Yaskawa INFORM job: OK_R2_O34(P)(180,90)OKKR.JBI

/JOB
//NAME OK_R2_O34(P)(180,90)OKKR
///FOLDERNAME X4
//POS
///NPOS 169,169,169,10,0,0
///TOOL 0
///POSTYPE PULSE
///PULSE
C00000=-166198,-138144,-82480,-6370,52509,85895
C00001=-166198,-138144,-82480,-6370,52509,85895
C00002=-181117,-122681,-70821,-2391,52511,79976
C00003=-181117,-121299,-68978,-2404,52087,79986
C00004=-181117,-122681,-70821,-2391,52511,79976
C00005=-189750,-118853,-70881,1473,64532,76480
C00006=-190053,-120746,-70880,1514,63564,76360
C00007=-189750,-118853,-70881,1473,64532,76480
C00008=-189574,-119616,-72884,1448,65370,76553
C00009=-189152,-121343,-77794,1387,67496,76728
C00010=-185679,-117174,-91161,1016,77811,78037
C00011=-185951,-117066,-86971,1049,75292,77923
C00012=-186063,-116900,-85242,1063,74315,77875
C00013=-185963,-114657,-82563,1057,73818,77905
C00014=-186063,-116900,-85242,1063,74315,77875
C00015=-189745,-129542,-86508,1430,68655,76533
C00016=-190220,-131942,-86638,1484,67510,76354
C00017=-189745,-129542,-86508,1430,68655,76533
C00018=-189571,-130130,-88400,1406,69515,76605
C00019=-189152,-131370,-93030,1352,71719,76776
C00020=-186714,-125767,-101679,2828,70067,77519
C00021=-186815,-124081,-96932,2888,68019,77434
C00022=-186348,-121871,-95196,2777,68068,77605
C00023=-186348,-120596,-92866,2792,67290,77587
C00024=-186348,-121871,-95196,2777,68068,77605
C00025=-189400,-136727,-97452,3651,61954,76311
C00026=-189193,-138074,-96714,3640,60801,76351
C00027=-189400,-136727,-97452,3651,61954,76311
C00028=-188527,-137172,-98533,3430,62352,76650
C00029=-188394,-140146,-103663,3351,63973,76748
C00030=-205862,-111673,-97339,6868,75787,70984
C00031=-186550,-124540,-97192,2829,67933,77528
C00032=-186590,-123775,-95257,2853,67137,77494
C00033=-186478,-121948,-93528,2830,67009,77531
C00034=-186590,-123775,-95257,2853,67137,77494
C00035=-188399,-134884,-95960,3412,61939,76686
C00036=-188879,-137801,-96233,3570,60632,76465
C00037=-188399,-134884,-95960,3412,61939,76686
C00038=-188346,-136077,-98025,3379,62594,76725
C00039=-188215,-138975,-103137,3302,64243,76822
C00040=-204668,-125654,-103075,12731,76819,72583
C00041=-192085,-108894,-77492,34918,79459,78781
C00042=-188431,-109256,-74124,35205,76110,79208
C00043=-186907,-109255,-72716,35331,74778,79404
C00044=-186693,-106850,-70345,35364,74503,79405
C00045=-186907,-109255,-72716,35331,74778,79404
C00046=-188549,-120012,-73127,36179,71120,77489
C00047=-189163,-122031,-72881,36386,70400,76982
C00048=-188549,-120012,-73127,36179,71120,77489
C00049=-190319,-120259,-74660,35963,72503,77227
C00050=-194524,-120520,-78356,35450,75955,76649
C00051=-198919,-109995,-61190,42638,67655,70810
C00052=-190285,-110618,-59420,40336,62273,73169
C00053=-188753,-109213,-57500,40420,61811,73628
C00054=-188509,-106588,-54755,40535,61445,73582
C00055=-188753,-109213,-57500,40420,61811,73628
C00056=-188387,-108235,-55987,37151,67409,76240
C00057=-189079,-110340,-56039,37365,66843,75742
C00058=-188387,-108235,-55987,37151,67409,76240
C00059=-190169,-108675,-57643,36861,68766,75986
C00060=-194403,-109476,-61648,36169,72132,75416
C00061=-225594,-162129,-113087,31828,88019,68030
C00062=-139895,-75891,-115387,-4844,89852,-32669
C00063=-106959,-65294,-90716,-19296,63371,-70213
C00064=-120633,-142199,-78464,-12,37387,-81752
C00065=-120609,-138941,-73010,-25,35704,-81740
C00066=-120602,-137609,-70801,-31,35029,-81735
C00067=-120604,-135014,-68605,-30,35012,-81736
C00068=-120602,-137609,-70801,-31,35029,-81735
C00069=-120446,-129838,-71958,-24,53874,-81685
C00070=-120438,-131177,-71579,-25,52953,-81682
C00071=-120446,-129838,-71958,-24,53874,-81685
C00072=-131738,-132228,-73452,8067,51560,-87163
C00073=-139177,-145158,-85992,13671,51481,-90607
C00074=-120880,-115298,-90682,38,78334,-81839
C00075=-120874,-115322,-86545,38,75775,-81838
C00076=-120876,-117328,-85486,38,74093,-81838
C00077=-120874,-115144,-83188,38,73801,-81838
C00078=-120876,-117328,-85486,38,74093,-81838
C00079=-120239,-131127,-87989,-18,68542,-81617
C00080=-120200,-135397,-88149,-23,66446,-81603
C00081=-120239,-131127,-87989,-18,68542,-81617
C00082=-120250,-131705,-89876,-17,69407,-81621
C00083=-120275,-132914,-94493,-15,71627,-81630
C00084=-120870,-123802,-101141,29,70454,-81834
C00085=-120864,-122259,-96439,28,68353,-81832
C00086=-120864,-123447,-95607,27,67230,-81833
C00087=-120862,-121131,-93340,27,67025,-81832
C00088=-120864,-123447,-95607,27,67230,-81833
C00089=-122761,-109093,-90522,1639,82538,-82345
C00090=-122816,-111754,-90455,1648,81130,-82381
C00091=-122761,-109093,-90522,1639,82538,-82345
C00092=-120406,-97391,-87876,-7,91529,-81675
C00093=-120406,-100930,-93432,-13,91808,-81675
C00094=-120586,-133914,-102382,9547,85095,-1839
C00095=-120585,-130719,-97494,9563,83747,-1942
C00096=-121451,-155216,-100429,10564,64059,-3872
C00097=-120574,-132034,-95782,9591,82039,-2069
C00098=-120583,-131496,-97319,9570,83246,-1979
C00099=-101302,-152747,-99963,8345,62763,3312
C00100=-120585,-128649,-94311,19028,83925,-4078
C00101=-120586,-131726,-99006,19000,85165,-3884
C00102=-120584,-126515,-91053,9592,81967,-2078
C00103=-120583,-123236,-86048,9622,80591,-2184
C00104=-121323,-131959,-83025,11198,58345,-4395
C00105=-120572,-124091,-84174,9663,79018,-2303
C00106=-120581,-123849,-85824,9632,80143,-2218
C00107=-103313,-130201,-82619,7208,57008,2414
C00108=-104272,-134854,-85867,7955,57176,1910
C00109=-120583,-124266,-87596,19086,82143,-4357
C00110=-121487,-140866,-77356,12448,52400,-5292
C00111=-120447,-141800,-70609,13740,42943,-6005
C00112=-120557,-138216,-68435,13384,45148,-5776
C00113=-120569,-112606,-67195,9826,74534,-2658
C00114=-120578,-112690,-68999,9781,75586,-2576
C00115=-93586,-136115,-68174,5406,43260,5492
C00116=-92921,-144795,-73490,5308,42038,5703
C00117=-124561,-133641,-73213,24753,58902,-8707
C00118=-106959,-65294,-90716,-19296,63371,-70213
C00119=-139895,-75891,-115387,-4844,89852,-32669
C00120=-225594,-162129,-113087,31828,88019,68030
C00121=-179306,-113082,-59158,46822,53733,18344
C00122=-185426,-123846,-62062,47213,53042,4581
C00123=-178966,-109306,-51351,46489,50599,6676
C00124=-174320,-104192,-54351,40123,55740,30099
C00125=-174328,-104480,-56277,39686,56549,30457
C00126=-160513,-108482,-51153,43765,42263,12341
C00127=-163416,-122959,-61489,45174,42800,10900
C00128=-171485,-113063,-58167,48901,53583,17150
C00129=-174246,-118964,-79181,37262,61787,32648
C00130=-175314,-125675,-85082,29507,69100,6827
C00131=-172538,-123885,-72027,36900,51897,2976
C00132=-174245,-116047,-71991,38244,59447,31724
C00133=-174254,-116050,-73753,37868,60313,32068
C00134=-155711,-121999,-71583,32332,45981,9052
C00135=-157559,-134878,-79454,33856,45162,7759
C00136=-184822,-140786,-87725,38201,57754,-504
C00137=-174185,-126575,-90838,36294,64403,33652
C00138=-184546,-129565,-98731,33104,80671,8257
C00139=-172470,-130384,-85545,34125,57897,8623
C00140=-174183,-124125,-83946,37166,61986,32753
C00141=-174193,-123890,-85598,36821,62909,33098
C00142=-156624,-128212,-85008,30161,52691,14183
C00143=-158543,-145659,-95435,31710,51171,12758
C00144=-172584,-141042,-104059,24276,66357,13202
C00145=-174271,-134419,-102558,-9435,85095,2061
C00146=-174282,-131199,-97661,-9450,83752,2158
C00147=-164002,-160404,-98949,-17577,58586,9036
C00148=-174285,-131975,-97483,-9458,83250,2195
C00149=-174277,-132508,-95944,-9478,82045,2290
C00150=-187249,-159818,-98857,-14082,54575,657
C00151=-174172,-139478,-100543,-16924,80978,4815
C00152=-174270,-132235,-99253,-18877,85281,4097
C00153=-174331,-126988,-91193,-9482,81954,2278
C00154=-155939,-119712,-87863,-13482,83832,9313
C00155=-158672,-128715,-82609,-15704,65966,9091
C00156=-174346,-124299,-85953,-9522,80133,2412
C00157=-174339,-124536,-84301,-9552,79010,2501
C00158=-176166,-130256,-82976,-13742,62349,3087
C00159=-165849,-135350,-93004,-16350,73762,7142
C00160=-174331,-124753,-87812,-18965,82235,4549
C00161=-174405,-116101,-74598,-9605,77388,2605
C00162=-166751,-128810,-77158,-12073,63289,6016
C00163=-170397,-124501,-65427,-14011,49451,5614
C00164=-174420,-113094,-69082,-9672,75561,2744
C00165=-174415,-113004,-67275,-9716,74511,2829
C00166=-190761,-123182,-65160,-8225,47369,-2619
C00167=-190350,-134813,-72783,-8527,46136,-2334
C00168=-168158,-141495,-72172,-29255,50267,11505
BC00000=196804,892977,1075175
BC00001=196804,892977,1075175
BC00002=196804,892977,1075175
BC00003=196804,892977,1075175
BC00004=196804,892977,1075175
BC00005=196804,892977,1075175
BC00006=196804,892977,1075175
BC00007=196804,892977,1075175
BC00008=196804,892977,1075175
BC00009=196804,892977,1075175
BC00010=223883,863738,1075175
BC00011=223883,863738,1075175
BC00012=223883,863738,1075175
BC00013=223883,863738,1075175
BC00014=223883,863738,1075175
BC00015=223883,863738,1075175
BC00016=223883,863738,1075175
BC00017=223883,863738,1075175
BC00018=223883,863738,1075175
BC00019=223883,863738,1075175
BC00020=258179,822666,1075175
BC00021=258179,822666,1075175
BC00022=258179,822666,1075175
BC00023=258179,822666,1075175
BC00024=258179,822666,1075175
BC00025=258179,822666,1075175
BC00026=258179,822666,1075175
BC00027=258179,822666,1075175
BC00028=258179,822666,1075175
BC00029=258179,822666,1075175
BC00030=349124,897467,1075175
BC00031=349124,897467,1075175
BC00032=349124,897467,1075175
BC00033=349124,897467,1075175
BC00034=349124,897467,1075175
BC00035=349124,897467,1075175
BC00036=349124,897467,1075175
BC00037=349124,897467,1075175
BC00038=349124,897467,1075175
BC00039=349124,897467,1075175
BC00040=330638,897048,1075175
BC00041=270427,895682,1075175
BC00042=270427,895682,1075175
BC00043=270427,895682,1075175
BC00044=270427,895682,1075175
BC00045=270427,895682,1075175
BC00046=270427,895682,1075175
BC00047=270427,895682,1075175
BC00048=270427,895682,1075175
BC00049=270427,895682,1075175
BC00050=270427,895682,1075175
BC00051=244019,926301,1075175
BC00052=244019,926301,1075175
BC00053=244019,926301,1075175
BC00054=244019,926301,1075175
BC00055=244019,926301,1075175
BC00056=244019,926301,1075175
BC00057=244019,926301,1075175
BC00058=244019,926301,1075175
BC00059=244019,926301,1075175
BC00060=244019,926301,1075175
BC00061=244019,926301,1075175
BC00062=284621,806624,1075175
BC00063=300201,760702,1075175
BC00064=369544,946445,1075175
BC00065=369544,946445,1075175
BC00066=369544,946445,1075175
BC00067=369544,946445,1075175
BC00068=369544,946445,1075175
BC00069=369544,946445,1075175
BC00070=369544,946445,1075175
BC00071=369544,946445,1075175
BC00072=369544,946445,1075175
BC00073=369544,946445,1075175
BC00074=370687,905748,1075175
BC00075=370687,905748,1075175
BC00076=370687,905748,1075175
BC00077=370687,905748,1075175
BC00078=370687,905748,1075175
BC00079=370687,905748,1075175
BC00080=370687,905748,1075175
BC00081=370687,905748,1075175
BC00082=370687,905748,1075175
BC00083=370687,905748,1075175
BC00084=370814,852872,1075175
BC00085=370814,852872,1075175
BC00086=370814,852872,1075175
BC00087=370814,852872,1075175
BC00088=370814,852872,1075175
BC00089=370814,852872,1075175
BC00090=370814,852872,1075175
BC00091=370814,852872,1075175
BC00092=370814,852872,1075175
BC00093=370814,852872,1075175
BC00094=333496,876256,1075175
BC00095=334875,878803,1075175
BC00096=335207,879415,1075175
BC00097=335427,879822,1075175
BC00098=335427,879822,1075175
BC00099=335207,879415,1075175
BC00100=332127,880440,1075175
BC00101=329407,878005,1075175
BC00102=333395,910749,1075175
BC00103=334774,913297,1075175
BC00104=335251,892678,1075175
BC00105=335326,914316,1075175
BC00106=335326,914316,1075175
BC00107=335251,892678,1075175
BC00108=335146,893402,1075175
BC00109=329306,912498,1075175
BC00110=333280,950895,1075175
BC00111=334659,953443,1075175
BC00112=334790,953685,1075175
BC00113=335211,954462,1075175
BC00114=335211,954462,1075175
BC00115=334790,953685,1075175
BC00116=334790,953685,1075175
BC00117=329191,952645,1075175
BC00118=300201,760702,1075175
BC00119=284621,806624,1075175
BC00120=244019,926301,1075175
BC00121=252810,904839,1075175
BC00122=251930,908762,1075175
BC00123=251930,908762,1075175
BC00124=251930,908762,1075175
BC00125=251930,908762,1075175
BC00126=251930,908762,1075175
BC00127=251930,908762,1075175
BC00128=250378,907547,1075175
BC00129=279615,874170,1075175
BC00130=278758,877989,1075175
BC00131=278758,877989,1075175
BC00132=278735,878093,1075175
BC00133=278735,878093,1075175
BC00134=278758,877989,1075175
BC00135=278758,877989,1075175
BC00136=278758,877989,1075175
BC00137=302654,847819,1075175
BC00138=301842,851437,1075175
BC00139=301842,851437,1075175
BC00140=301773,851742,1075175
BC00141=301773,851742,1075175
BC00142=301842,851437,1075175
BC00143=301842,851437,1075175
BC00144=301842,851437,1075175
BC00145=254856,848220,1075175
BC00146=252114,849302,1075175
BC00147=251037,849726,1075175
BC00148=251017,849734,1075175
BC00149=251017,849734,1075175
BC00150=251037,849726,1075175
BC00151=251037,849726,1075175
BC00152=256865,852098,1075175
BC00153=231817,874571,1075175
BC00154=231101,858363,1075175
BC00155=231101,858363,1075175
BC00156=227978,876085,1075175
BC00157=227978,876085,1075175
BC00158=231101,858363,1075175
BC00159=231101,858363,1075175
BC00160=233826,878449,1075175
BC00161=205012,905240,1075175
BC00162=209704,892317,1075175
BC00163=209704,892317,1075175
BC00164=201173,906754,1075175
BC00165=201173,906754,1075175
BC00166=209704,892317,1075175
BC00167=209704,892317,1075175
BC00168=207022,909118,1075175
EC00000=1596313,309153
EC00001=1596313,309153
EC00002=1596313,309153
EC00003=1596313,309153
EC00004=1596313,309153
EC00005=1596313,309153
EC00006=1596313,309153
EC00007=1596313,309153
EC00008=1596313,309153
EC00009=1596313,309153
EC00010=1596313,309153
EC00011=1596313,309153
EC00012=1596313,309153
EC00013=1596313,309153
EC00014=1596313,309153
EC00015=1596313,309153
EC00016=1596313,309153
EC00017=1596313,309153
EC00018=1596313,309153
EC00019=1596313,309153
EC00020=1596313,309153
EC00021=1596313,309153
EC00022=1596313,309153
EC00023=1596313,309153
EC00024=1596313,309153
EC00025=1596313,309153
EC00026=1596313,309153
EC00027=1596313,309153
EC00028=1596313,309153
EC00029=1596313,309153
EC00030=1596313,309153
EC00031=1596313,309153
EC00032=1596313,309153
EC00033=1596313,309153
EC00034=1596313,309153
EC00035=1596313,309153
EC00036=1596313,309153
EC00037=1596313,309153
EC00038=1596313,309153
EC00039=1596313,309153
EC00040=1596313,309153
EC00041=1596313,309153
EC00042=1596313,309153
EC00043=1596313,309153
EC00044=1596313,309153
EC00045=1596313,309153
EC00046=1596313,309153
EC00047=1596313,309153
EC00048=1596313,309153
EC00049=1596313,309153
EC00050=1596313,309153
EC00051=1596313,309153
EC00052=1596313,309153
EC00053=1596313,309153
EC00054=1596313,309153
EC00055=1596313,309153
EC00056=1596313,309153
EC00057=1596313,309153
EC00058=1596313,309153
EC00059=1596313,309153
EC00060=1596313,309153
EC00061=1596313,309153
EC00062=1596313,494645
EC00063=1596313,556475
EC00064=1596313,556475
EC00065=1596313,556475
EC00066=1596313,556475
EC00067=1596313,556475
EC00068=1596313,556475
EC00069=1596313,556475
EC00070=1596313,556475
EC00071=1596313,556475
EC00072=1596313,556475
EC00073=1596313,556475
EC00074=1596313,556475
EC00075=1596313,556475
EC00076=1596313,556475
EC00077=1596313,556475
EC00078=1596313,556475
EC00079=1596313,556475
EC00080=1596313,556475
EC00081=1596313,556475
EC00082=1596313,556475
EC00083=1596313,556475
EC00084=1596313,556475
EC00085=1596313,556475
EC00086=1596313,556475
EC00087=1596313,556475
EC00088=1596313,556475
EC00089=1596313,556475
EC00090=1596313,556475
EC00091=1596313,556475
EC00092=1596313,556475
EC00093=1596313,556475
EC00094=1596313,556475
EC00095=1596313,556475
EC00096=1596313,556475
EC00097=1596313,556475
EC00098=1596313,556475
EC00099=1596313,556475
EC00100=1596313,556475
EC00101=1596313,556475
EC00102=1596313,556475
EC00103=1596313,556475
EC00104=1596313,556475
EC00105=1596313,556475
EC00106=1596313,556475
EC00107=1596313,556475
EC00108=1596313,556475
EC00109=1596313,556475
EC00110=1596313,556475
EC00111=1596313,556475
EC00112=1596313,556475
EC00113=1596313,556475
EC00114=1596313,556475
EC00115=1596313,556475
EC00116=1596313,556475
EC00117=1596313,556475
EC00118=1596313,556475
EC00119=1596313,494645
EC00120=1596313,309153
EC00121=1596313,309153
EC00122=1596313,309153
EC00123=1596313,309153
EC00124=1596313,309153
EC00125=1596313,309153
EC00126=1596313,309153
EC00127=1596313,309153
EC00128=1596313,309153
EC00129=1596313,309153
EC00130=1596313,309153
EC00131=1596313,309153
EC00132=1596313,309153
EC00133=1596313,309153
EC00134=1596313,309153
EC00135=1596313,309153
EC00136=1596313,309153
EC00137=1596313,309153
EC00138=1596313,309153
EC00139=1596313,309153
EC00140=1596313,309153
EC00141=1596313,309153
EC00142=1596313,309153
EC00143=1596313,309153
EC00144=1596313,309153
EC00145=1596313,309153
EC00146=1596313,309153
EC00147=1596313,309153
EC00148=1596313,309153
EC00149=1596313,309153
EC00150=1596313,309153
EC00151=1596313,309153
EC00152=1596313,309153
EC00153=1596313,309153
EC00154=1596313,309153
EC00155=1596313,309153
EC00156=1596313,309153
EC00157=1596313,309153
EC00158=1596313,309153
EC00159=1596313,309153
EC00160=1596313,309153
EC00161=1596313,309153
EC00162=1596313,309153
EC00163=1596313,309153
EC00164=1596313,309153
EC00165=1596313,309153
EC00166=1596313,309153
EC00167=1596313,309153
EC00168=1596313,309153
///POSTYPE BASE
///RECTAN
///RCONF 0,0,0,0,0,0,0,0,0,0,0,0,0,0,0,0,0,0,0,0,0,0,0,0
P00006=0.222,-3.123,-1.508,0.0000,0.0000,0.0000
P00021=-0.225,-6.128,-0.405,0.0000,0.0000,0.0000
P00022=0.222,-3.123,-1.508,0.0000,0.0000,0.0000
P00023=0.143,-0.036,0.682,0.0000,0.0000,0.0000
P00031=1.853,-0.001,-1.549,0.0000,0.0000,0.0000
P00032=1.957,0.503,-7.217,0.0000,0.0000,0.0000
///RCONF 0,0,0,0,1,0,0,0,0,0,0,0,0,0,0,0,0,0,0,0,0,0,0,0
P00033=-0.123,0.612,-5.012,0.0000,0.0000,0.0000
///RCONF 0,0,0,0,0,0,0,0,0,0,0,0,0,0,0,0,0,0,0,0,0,0,0,0
P00041=0.192,3.924,0.305,0.0000,0.0000,0.0000
P00042=-0.217,1.941,0.413,0.0000,0.0000,0.0000
P00043=-0.044,-1.937,1.197,0.0000,0.0000,0.0000
//INST
///DATE 2023/12/13 11:22
///ATTR SC,RW
///GROUP1 RB1,BS1
///GROUP2 ST1
NOP
'OK_r2_O34(P)(180,90)
'180,50
'Path S1834
SFTOF3D
MOVJ C00000 BC00000 VJ=100.00  +MOVJ EC00000 VJ=100.00
MOVL C00001 BC00001 V=400.0  +MOVJ EC00001 VJ=100.00
SMOVL C00002 BC00002 V=60.0  +MOVJ EC00002
SREFP 3 C00003 BC00003  +REFP EC00003
CALL JOB:SEARCH-R1-S13D
SET P041 P006
SFTON3D P041
SMOVL C00004 BC00004 V=60.0  +MOVJ EC00004
SMOVL C00005 BC00005 V=60.0  +MOVJ EC00005
SREFP 3 C00006 BC00006  +REFP EC00006
CALL JOB:SEARCH-R1-S13D
SET P041 P006
SFTON3D P041
SMOVL C00007 BC00007 V=60.0  +MOVJ EC00007
MOVL C00008 BC00008 V=400.0  +MOVJ EC00008 VJ=100.00
MOVL C00009 BC00009 V=1000.0  +MOVJ EC00009 VJ=100.00
'Path S1835
SFTOF3D
MOVJ C00010 BC00010 VJ=100.00  +MOVJ EC00010 VJ=100.00
MOVL C00011 BC00011 V=400.0  +MOVJ EC00011 VJ=100.00
SMOVL C00012 BC00012 V=60.0  +MOVJ EC00012
SREFP 3 C00013 BC00013  +REFP EC00013
CALL JOB:SEARCH-R1-S13D
SET P042 P006
SFTON3D P042
SMOVL C00014 BC00014 V=60.0  +MOVJ EC00014
SMOVL C00015 BC00015 V=60.0  +MOVJ EC00015
SREFP 3 C00016 BC00016  +REFP EC00016
CALL JOB:SEARCH-R1-S13D
SET P042 P006
SFTON3D P042
SMOVL C00017 BC00017 V=60.0  +MOVJ EC00017
MOVL C00018 BC00018 V=400.0  +MOVJ EC00018 VJ=100.00
MOVL C00019 BC00019 V=1000.0  +MOVJ EC00019 VJ=100.00
'Path S1836
SFTOF3D
MOVJ C00020 BC00020 VJ=100.00  +MOVJ EC00020 VJ=100.00
MOVL C00021 BC00021 V=400.0  +MOVJ EC00021 VJ=100.00
SMOVL C00022 BC00022 V=60.0  +MOVJ EC00022
SREFP 3 C00023 BC00023  +REFP EC00023
CALL JOB:SEARCH-R1-S13D
SET P043 P006
SFTON3D P043
SMOVL C00024 BC00024 V=60.0  +MOVJ EC00024
SMOVL C00025 BC00025 V=60.0  +MOVJ EC00025
SREFP 3 C00026 BC00026  +REFP EC00026
CALL JOB:SEARCH-R1-S13D
SET P043 P006
SFTON3D P043
SMOVL C00027 BC00027 V=60.0  +MOVJ EC00027
MOVL C00028 BC00028 V=400.0  +MOVJ EC00028 VJ=100.00
MOVL C00029 BC00029 V=1000.0  +MOVJ EC00029 VJ=100.00
'Path S1830
SFTOF3D
MOVJ C00030 BC00030 VJ=100.00  +MOVJ EC00030 VJ=100.00
MOVL C00031 BC00031 V=400.0  +MOVJ EC00031 VJ=100.00
SMOVL C00032 BC00032 V=60.0  +MOVJ EC00032
SREFP 3 C00033 BC00033  +REFP EC00033
CALL JOB:SEARCH-R1-S13D
SET P033 P006
SFTON3D P033
SMOVL C00034 BC00034 V=60.0  +MOVJ EC00034
SMOVL C00035 BC00035 V=60.0  +MOVJ EC00035
SREFP 3 C00036 BC00036  +REFP EC00036
CALL JOB:SEARCH-R1-S13D
SET P033 P006
SFTON3D P033
SMOVL C00037 BC00037 V=60.0  +MOVJ EC00037
MOVL C00038 BC00038 V=400.0  +MOVJ EC00038 VJ=100.00
MOVL C00039 BC00039 V=1000.0  +MOVJ EC00039 VJ=100.00
'Path S1829
SFTOF3D
MOVJ C00040 BC00040 VJ=20.00  +MOVJ EC00040 VJ=0.78
MOVJ C00041 BC00041 VJ=100.00  +MOVJ EC00041 VJ=100.00
MOVL C00042 BC00042 V=400.0  +MOVJ EC00042 VJ=100.00
SMOVL C00043 BC00043 V=60.0  +MOVJ EC00043
SREFP 3 C00044 BC00044  +REFP EC00044
CALL JOB:SEARCH-R1-S13D
SET P032 P006
SFTON3D P032
SMOVL C00045 BC00045 V=60.0  +MOVJ EC00045
SMOVL C00046 BC00046 V=60.0  +MOVJ EC00046
SREFP 3 C00047 BC00047  +REFP EC00047
CALL JOB:SEARCH-R1-S13D
SET P032 P006
SFTON3D P032
SMOVL C00048 BC00048 V=60.0  +MOVJ EC00048
MOVL C00049 BC00049 V=400.0  +MOVJ EC00049 VJ=100.00
MOVL C00050 BC00050 V=1000.0  +MOVJ EC00050 VJ=100.00
'Path S1828
SFTOF3D
MOVJ C00051 BC00051 VJ=100.00  +MOVJ EC00051 VJ=100.00
MOVL C00052 BC00052 V=400.0  +MOVJ EC00052 VJ=100.00
SMOVL C00053 BC00053 V=60.0  +MOVJ EC00053
SREFP 3 C00054 BC00054  +REFP EC00054
CALL JOB:SEARCH-R1-S13D
SET P031 P006
SFTON3D P031
SMOVL C00055 BC00055 V=60.0  +MOVJ EC00055
SMOVL C00056 BC00056 V=60.0  +MOVJ EC00056
SREFP 3 C00057 BC00057  +REFP EC00057
CALL JOB:SEARCH-R1-S13D
SET P031 P006
SFTON3D P031
SMOVL C00058 BC00058 V=60.0  +MOVJ EC00058
MOVL C00059 BC00059 V=400.0  +MOVJ EC00059 VJ=100.00
MOVL C00060 BC00060 V=1000.0  +MOVJ EC00060 VJ=100.00
MOVJ C00061 BC00061 VJ=100.00  +MOVJ EC00061 VJ=100.00
MOVJ C00062 BC00062 VJ=100.00  +MOVJ EC00062 VJ=100.00
MOVJ C00063 BC00063 VJ=100.00  +MOVJ EC00063 VJ=100.00
'180,0
'Path S1083
SFTOF3D
MOVJ C00064 BC00064 VJ=100.00  +MOVJ EC00064 VJ=100.00
MOVL C00065 BC00065 V=400.0  +MOVJ EC00065 VJ=100.00
SMOVL C00066 BC00066 V=60.0  +MOVJ EC00066
SREFP 3 C00067 BC00067  +REFP EC00067
CALL JOB:SEARCH-R1-S13D
SET P021 P006
SFTON3D P021
SMOVL C00068 BC00068 V=60.0  +MOVJ EC00068
SMOVL C00069 BC00069 V=60.0  +MOVJ EC00069
SREFP 3 C00070 BC00070  +REFP EC00070
CALL JOB:SEARCH-R1-S13D
SET P021 P006
SFTON3D P021
SMOVL C00071 BC00071 V=60.0  +MOVJ EC00071
MOVL C00072 BC00072 V=400.0  +MOVJ EC00072 VJ=100.00
MOVL C00073 BC00073 V=1000.0  +MOVJ EC00073 VJ=100.00
'Path S1084
SFTOF3D
MOVJ C00074 BC00074 VJ=100.00  +MOVJ EC00074 VJ=100.00
MOVL C00075 BC00075 V=400.0  +MOVJ EC00075 VJ=100.00
SMOVL C00076 BC00076 V=60.0  +MOVJ EC00076
SREFP 3 C00077 BC00077  +REFP EC00077
CALL JOB:SEARCH-R1-S13D
SET P022 P006
SFTON3D P022
SMOVL C00078 BC00078 V=60.0  +MOVJ EC00078
SMOVL C00079 BC00079 V=60.0  +MOVJ EC00079
SREFP 3 C00080 BC00080  +REFP EC00080
CALL JOB:SEARCH-R1-S13D
SET P022 P006
SFTON3D P022
SMOVL C00081 BC00081 V=60.0  +MOVJ EC00081
MOVL C00082 BC00082 V=400.0  +MOVJ EC00082 VJ=100.00
MOVL C00083 BC00083 V=1000.0  +MOVJ EC00083 VJ=100.00
'Path S1085
SFTOF3D
MOVJ C00084 BC00084 VJ=100.00  +MOVJ EC00084 VJ=100.00
MOVL C00085 BC00085 V=400.0  +MOVJ EC00085 VJ=100.00
SMOVL C00086 BC00086 V=60.0  +MOVJ EC00086
SREFP 3 C00087 BC00087  +REFP EC00087
CALL JOB:SEARCH-R1-S13D
SET P023 P006
SFTON3D P023
SMOVL C00088 BC00088 V=60.0  +MOVJ EC00088
SMOVL C00089 BC00089 V=60.0  +MOVJ EC00089
SREFP 3 C00090 BC00090  +REFP EC00090
CALL JOB:SEARCH-R1-S13D
SET P023 P006
SFTON3D P023
SMOVL C00091 BC00091 V=60.0  +MOVJ EC00091
MOVL C00092 BC00092 V=400.0  +MOVJ EC00092 VJ=100.00
MOVL C00093 BC00093 V=1000.0  +MOVJ EC00093 VJ=100.00
'Path W275
SFTOF3D
SFTON3D P023
MOVJ C00094 BC00094 VJ=100.00  +MOVJ EC00094 VJ=100.00
SMOVL C00095 BC00095 V=400.0  +MOVJ EC00095
SMOVL C00096 BC00096 V=100.0 PL=0  +MOVJ EC00096
SREFP 1 C00097 BC00097  +REFP EC00097
SREFP 2 C00098 BC00098  +REFP EC00098
MACRO1 MJ#(0) ARGF0
ARCON
SMOVL C00099 BC00099 V=10.0  +MOVJ EC00099
ARCOF
SMOVL C00100 BC00100 V=400.0  +MOVJ EC00100
SMOVL C00101 BC00101 V=1000.0  +MOVJ EC00101
SFTOF3D
'Path W276
SFTOF3D
SFTON3D P022
MOVJ C00102 BC00102 VJ=100.00  +MOVJ EC00102 VJ=100.00
SMOVL C00103 BC00103 V=400.0  +MOVJ EC00103
SMOVL C00104 BC00104 V=100.0 PL=0  +MOVJ EC00104
SREFP 1 C00105 BC00105  +REFP EC00105
SREFP 2 C00106 BC00106  +REFP EC00106
MACRO1 MJ#(0) ARGF0
ARCON
SMOVL C00107 BC00107 V=10.0  +MOVJ EC00107
ARCOF
SMOVL C00108 BC00108 V=400.0  +MOVJ EC00108
SMOVL C00109 BC00109 V=1000.0  +MOVJ EC00109
SFTOF3D
'Path W278
SFTOF3D
SFTON3D P021
MOVJ C00110 BC00110 VJ=100.00  +MOVJ EC00110 VJ=100.00
SMOVL C00111 BC00111 V=400.0  +MOVJ EC00111
SMOVL C00112 BC00112 V=100.0 PL=0  +MOVJ EC00112
SREFP 1 C00113 BC00113  +REFP EC00113
SREFP 2 C00114 BC00114  +REFP EC00114
MACRO1 MJ#(0) ARGF0
ARCON
SMOVL C00115 BC00115 V=10.0  +MOVJ EC00115
ARCOF
SMOVL C00116 BC00116 V=400.0  +MOVJ EC00116
SMOVL C00117 BC00117 V=1000.0  +MOVJ EC00117
SFTOF3D
MOVJ C00118 BC00118 VJ=100.00  +MOVJ EC00118 VJ=100.00
MOVJ C00119 BC00119 VJ=100.00  +MOVJ EC00119 VJ=100.00
MOVJ C00120 BC00120 VJ=100.00  +MOVJ EC00120 VJ=100.00
'180,50
'Path W1839
SFTOF3D
SFTON3D P031
MOVJ C00121 BC00121 VJ=100.00  +MOVJ EC00121 VJ=100.00
SMOVL C00122 BC00122 V=400.0  +MOVJ EC00122
SMOVL C00123 BC00123 V=100.0 PL=0  +MOVJ EC00123
SREFP 1 C00124 BC00124  +REFP EC00124
SREFP 2 C00125 BC00125  +REFP EC00125
MACRO1 MJ#(0) ARGF0
ARCON
SMOVL C00126 BC00126 V=10.0  +MOVJ EC00126
ARCOF
SMOVL C00127 BC00127 V=400.0  +MOVJ EC00127
SMOVL C00128 BC00128 V=1000.0  +MOVJ EC00128
SFTOF3D
'Path W1838
SFTOF3D
SFTON3D P032
MOVJ C00129 BC00129 VJ=100.00  +MOVJ EC00129 VJ=100.00
SMOVL C00130 BC00130 V=400.0  +MOVJ EC00130
SMOVL C00131 BC00131 V=100.0 PL=0  +MOVJ EC00131
SREFP 1 C00132 BC00132  +REFP EC00132
SREFP 2 C00133 BC00133  +REFP EC00133
MACRO1 MJ#(0) ARGF0
ARCON
SMOVL C00134 BC00134 V=10.0  +MOVJ EC00134
ARCOF
SMOVL C00135 BC00135 V=400.0  +MOVJ EC00135
SMOVL C00136 BC00136 V=1000.0  +MOVJ EC00136
SFTOF3D
'Path W1837
SFTOF3D
SFTON3D P033
MOVJ C00137 BC00137 VJ=100.00  +MOVJ EC00137 VJ=100.00
SMOVL C00138 BC00138 V=400.0  +MOVJ EC00138
SMOVL C00139 BC00139 V=100.0 PL=0  +MOVJ EC00139
SREFP 1 C00140 BC00140  +REFP EC00140
SREFP 2 C00141 BC00141  +REFP EC00141
MACRO1 MJ#(0) ARGF0
ARCON
SMOVL C00142 BC00142 V=10.0  +MOVJ EC00142
ARCOF
SMOVL C00143 BC00143 V=400.0  +MOVJ EC00143
SMOVL C00144 BC00144 V=1000.0  +MOVJ EC00144
SFTOF3D
'Path W1840
SFTOF3D
SFTON3D P043
MOVJ C00145 BC00145 VJ=100.00  +MOVJ EC00145 VJ=100.00
SMOVL C00146 BC00146 V=400.0  +MOVJ EC00146
SMOVL C00147 BC00147 V=100.0 PL=0  +MOVJ EC00147
SREFP 1 C00148 BC00148  +REFP EC00148
SREFP 2 C00149 BC00149  +REFP EC00149
MACRO1 MJ#(0) ARGF0
ARCON
SMOVL C00150 BC00150 V=10.0  +MOVJ EC00150
ARCOF
SMOVL C00151 BC00151 V=400.0  +MOVJ EC00151
SMOVL C00152 BC00152 V=1000.0  +MOVJ EC00152
SFTOF3D
'Path W1841
SFTOF3D
SFTON3D P042
MOVJ C00153 BC00153 VJ=100.00  +MOVJ EC00153 VJ=100.00
SMOVL C00154 BC00154 V=400.0  +MOVJ EC00154
SMOVL C00155 BC00155 V=100.0 PL=0  +MOVJ EC00155
SREFP 1 C00156 BC00156  +REFP EC00156
SREFP 2 C00157 BC00157  +REFP EC00157
MACRO1 MJ#(0) ARGF0
ARCON
SMOVL C00158 BC00158 V=10.0  +MOVJ EC00158
ARCOF
SMOVL C00159 BC00159 V=400.0  +MOVJ EC00159
SMOVL C00160 BC00160 V=1000.0  +MOVJ EC00160
SFTOF3D
'Path W1842
SFTOF3D
SFTON3D P041
MOVJ C00161 BC00161 VJ=100.00  +MOVJ EC00161 VJ=100.00
SMOVL C00162 BC00162 V=400.0  +MOVJ EC00162
SMOVL C00163 BC00163 V=100.0 PL=0  +MOVJ EC00163
SREFP 1 C00164 BC00164  +REFP EC00164
SREFP 2 C00165 BC00165  +REFP EC00165
MACRO1 MJ#(0) ARGF0
ARCON
SMOVL C00166 BC00166 V=10.0  +MOVJ EC00166
ARCOF
SMOVL C00167 BC00167 V=400.0  +MOVJ EC00167
SMOVL C00168 BC00168 V=1000.0  +MOVJ EC00168
SFTOF3D
END
